(* Schneider Machine Expert - Basic project Maquina, file version 2.9.0.0 *)
(* ProjectInformations: Name=Nuevo proyecto *)

HARDWARE
  Cpu 0: TM221CE16T
  EthernetConfiguration: NetworkName=M221, IpAllocationMode=FixedAddress, IpAddress=192.168.0.10, SubnetMask=255.255.255.0
  SerialLineConfiguration: Baud=Baud19200, Parity=ParityEven, DataBits=DataBits8, StopBits=StopBits1, PhysicalMedium=PhysicalMediumRs485, TransmissionMode=TransmissionModeModbusRtu, SlaveId=1, Addressing=SlaveAddressing
  MastTask: UsePeriodScanMode=false, PeriodScan=100
  FastTask: Period=255
  CpuBehavior: StartingMode=StartAsPreviousState, AutoSaveRamOnEeprom=true, WatchdogPeriod=250

SYMBOLS  (address, symbol, comment, settings)
  %M1       INICIO_MANUAL  "start Manual"
  %M2       INICIO_AUTOM  "Automatico"
  %M3       STOP
  %M4       AUT_ARRIBA
  %M5       RESET  "Nueva medicion"
  %M6       RESET_MANUAL  "reset manual"
  %M8       TIEM_MUESTREO_ON
  %M9       SUBIR
  %M10      BAJAR  "Bajar_manual"
  %M12      BAJAR_AUTO  "Hab.Pulsos"
  %M13      GRAFICA  "Hab.Grafica"
  %M14      AUTOMA_ON
  %M15      HA_AUTOMATICO
  %M16      MANUAL_ON
  %M17      HA_MANUAL
  %M18      AUT_ABAJO
  %M19      SUBIR_AUTO
  %M20      ESTADO1
  %M21      ESTADO2
  %M22      ESTADO3
  %M23      ESTADO4
  %MW2      VALOR_MENOR
  %MW3      VALOR_MAYOR
  %MW4      MAYOR
  %MW8      TIEMPO_MUESTREO
  %MW11     DATOSGRAFICA
  %KW0      ESCA  [Value=10]
  %TM1        [Preset=10, Base=OneMilliSeconds]
  %TM2        [Preset=10, Base=OneMilliSeconds]
  %TM3        [Preset=10, Base=OneMilliSeconds]
  %I0.1     SEN_INFERIOR
  %I0.3     SEN_SUPERIOR
  %Q0.2     SENGIRO
  %IW0.1    CELDA  [Type=Type_0_10V, Scope=Scope_Normal, Minimum=0, Maximum=1000]
  %FREQGEN0 MOTOR  [PtoObject(RefInput=NotUsed, ZPhaseInput=NotUsed, ProbeInput=NotUsed), GlobalIndex=0, Type=FREQGEN, Preset=1, SignalFrequency=2000]
  %FREQGEN1 DATOS  [PtoObject(RefInput=NotUsed, ZPhaseInput=NotUsed, ProbeInput=NotUsed), GlobalIndex=1, Type=FREQGEN, TimeBase=OneMilliSeconds, Preset=1, SignalFrequency=200]

POU Nuevo POU
  (* SectionNumber=1 *)

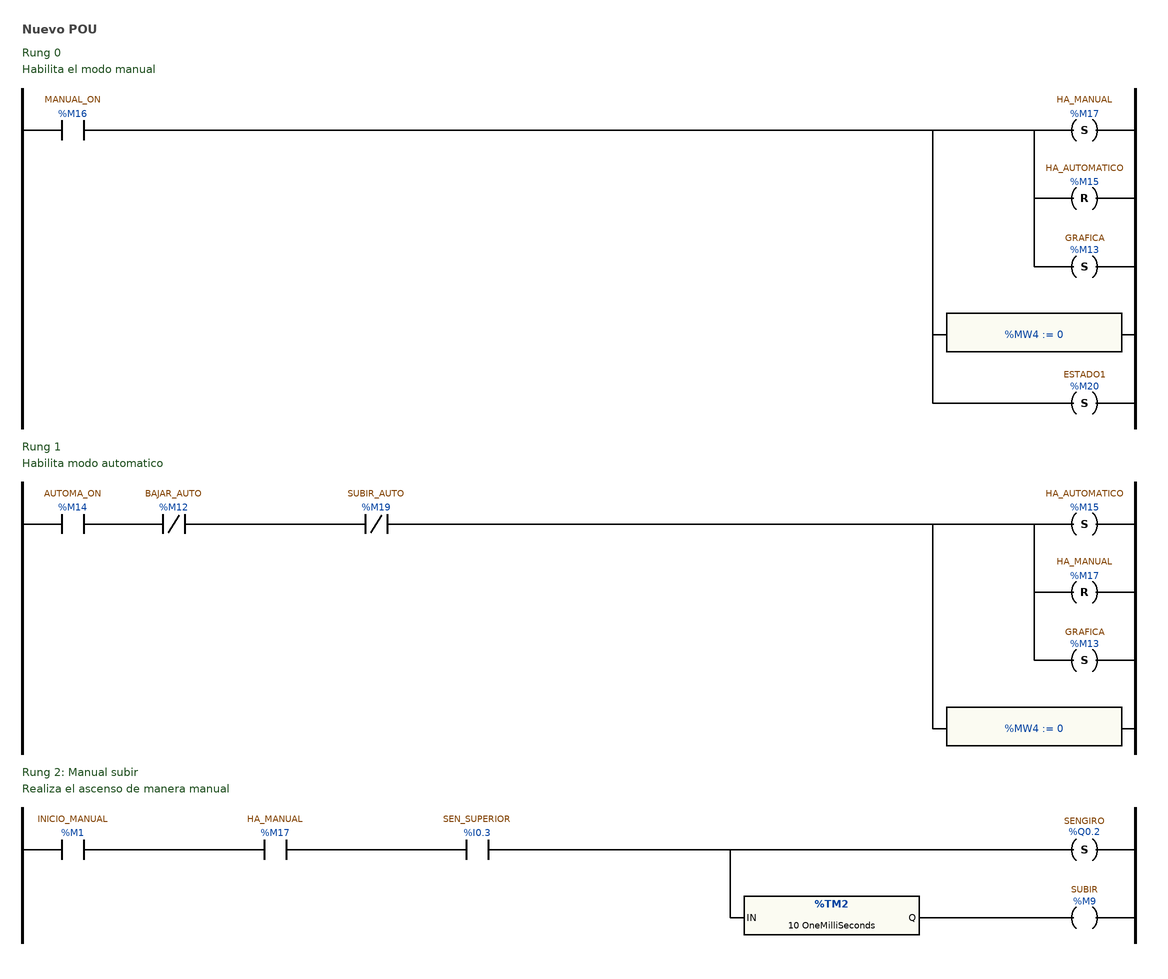

// Rung 0
// Habilita el modo manual
  LD %M16                 (* MANUAL_ON *)
  S %M17                  (* HA_MANUAL *)
  R %M15                  (* HA_AUTOMATICO *)
  S %M13                  (* GRAFICA *)
  [ %MW4 := 0 ]           (* MAYOR *)
  S %M20                  (* ESTADO1 *)
  // as ST:
  //   IF MANUAL_ON THEN HA_MANUAL := TRUE; END_IF;
  //   IF MANUAL_ON THEN HA_AUTOMATICO := FALSE; END_IF;
  //   IF MANUAL_ON THEN GRAFICA := TRUE; END_IF;
  //   IF MANUAL_ON THEN MAYOR := 0; END_IF;
  //   IF MANUAL_ON THEN ESTADO1 := TRUE; END_IF;

// Rung 1
// Habilita modo automatico
  LD %M14                 (* AUTOMA_ON *)
  ANDN %M12               (* BAJAR_AUTO *)
  ANDN %M19               (* SUBIR_AUTO *)
  S %M15                  (* HA_AUTOMATICO *)
  R %M17                  (* HA_MANUAL *)
  S %M13                  (* GRAFICA *)
  [ %MW4 := 0 ]           (* MAYOR *)
  // as ST:
  //   IF AUTOMA_ON AND NOT BAJAR_AUTO AND NOT SUBIR_AUTO THEN HA_AUTOMATICO := TRUE; END_IF;
  //   IF AUTOMA_ON AND NOT BAJAR_AUTO AND NOT SUBIR_AUTO THEN HA_MANUAL := FALSE; END_IF;
  //   IF AUTOMA_ON AND NOT BAJAR_AUTO AND NOT SUBIR_AUTO THEN GRAFICA := TRUE; END_IF;
  //   IF AUTOMA_ON AND NOT BAJAR_AUTO AND NOT SUBIR_AUTO THEN MAYOR := 0; END_IF;

// Rung 2: Manual subir
// Realiza el ascenso de manera manual
  LD 1
  MULTIFB
  LD 1
  AND %M1                 (* INICIO_MANUAL *)
  AND %M17                (* HA_MANUAL *)
  AND %I0.3               (* SEN_SUPERIOR *)
  ST %MW2009:X0
  LD %MW2009:X0
  S %Q0.2                 (* SENGIRO *)
  BLK %TM2
  LD %MW2009:X0
  IN
  OUT_BLK
  LD Q
  ST %M9                  (* SUBIR *)
  END_BLK
  MULTIFB
  // as ST:
  //   IF INICIO_MANUAL AND HA_MANUAL AND SEN_SUPERIOR THEN SENGIRO := TRUE; END_IF;
  //   %TM2(IN := INICIO_MANUAL AND HA_MANUAL AND SEN_SUPERIOR);
  //   SUBIR := %TM2.Q;

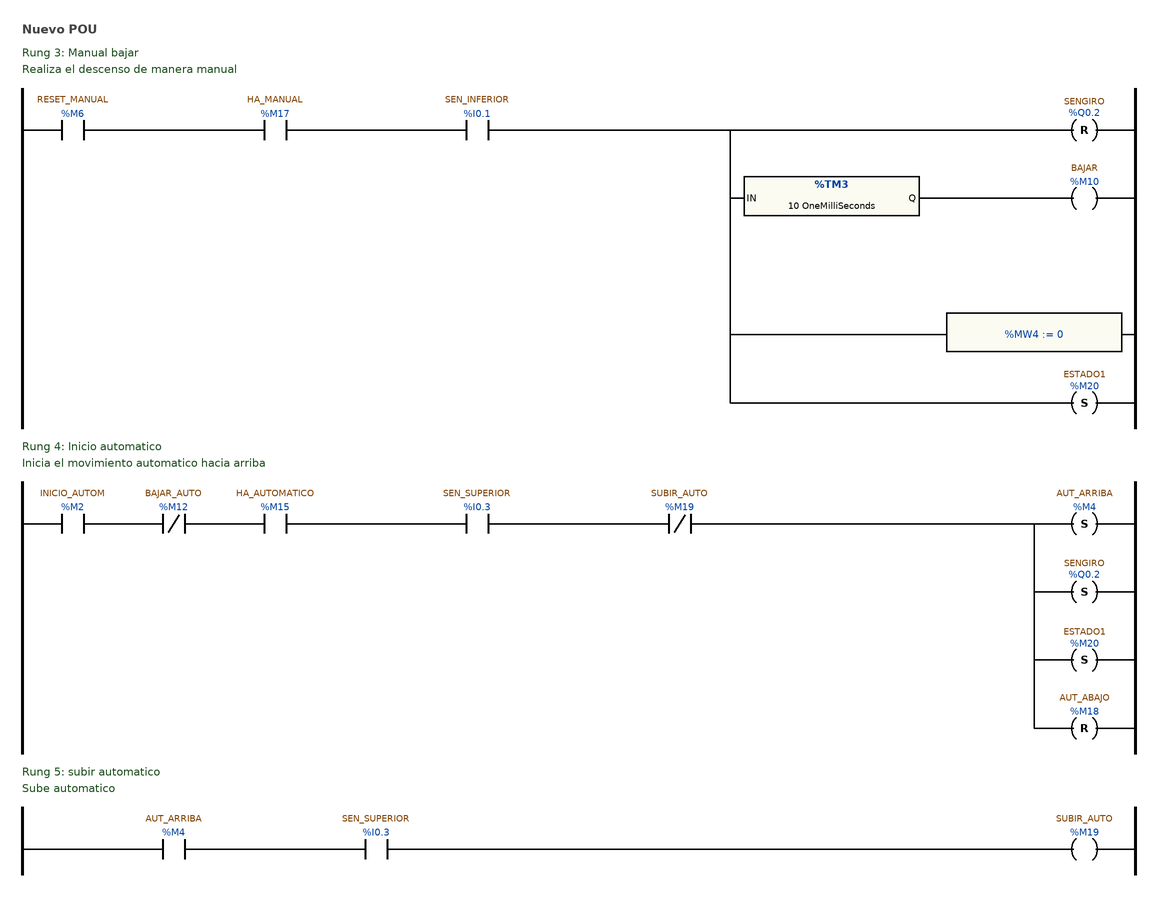

// Rung 3: Manual bajar
// Realiza el descenso de manera manual
  LD 1
  MULTIFB
  LD 1
  AND %M6                 (* RESET_MANUAL *)
  AND %M17                (* HA_MANUAL *)
  AND %I0.1               (* SEN_INFERIOR *)
  ST %MW2009:X0
  LD %MW2009:X0
  R %Q0.2                 (* SENGIRO *)
  BLK %TM3
  LD %MW2009:X0
  IN
  OUT_BLK
  LD Q
  ST %M10                 (* BAJAR *)
  END_BLK
  LD %MW2009:X0
  [ %MW4 := 0 ]           (* MAYOR *)
  S %M20                  (* ESTADO1 *)
  MULTIFB
  // as ST:
  //   IF RESET_MANUAL AND HA_MANUAL AND SEN_INFERIOR THEN SENGIRO := FALSE; END_IF;
  //   %TM3(IN := RESET_MANUAL AND HA_MANUAL AND SEN_INFERIOR);
  //   BAJAR := %TM3.Q;
  //   IF RESET_MANUAL AND HA_MANUAL AND SEN_INFERIOR THEN MAYOR := 0; END_IF;
  //   IF RESET_MANUAL AND HA_MANUAL AND SEN_INFERIOR THEN ESTADO1 := TRUE; END_IF;

// Rung 4: Inicio automatico
// Inicia el movimiento automatico hacia arriba
  LD %M2                  (* INICIO_AUTOM *)
  ANDN %M12               (* BAJAR_AUTO *)
  AND %M15                (* HA_AUTOMATICO *)
  AND %I0.3               (* SEN_SUPERIOR *)
  ANDN %M19               (* SUBIR_AUTO *)
  S %M4                   (* AUT_ARRIBA *)
  S %Q0.2                 (* SENGIRO *)
  S %M20                  (* ESTADO1 *)
  R %M18                  (* AUT_ABAJO *)
  // as ST:
  //   IF INICIO_AUTOM AND NOT BAJAR_AUTO AND HA_AUTOMATICO AND SEN_SUPERIOR AND NOT SUBIR_AUTO THEN AUT_ARRIBA := TRUE; END_IF;
  //   IF INICIO_AUTOM AND NOT BAJAR_AUTO AND HA_AUTOMATICO AND SEN_SUPERIOR AND NOT SUBIR_AUTO THEN SENGIRO := TRUE; END_IF;
  //   IF INICIO_AUTOM AND NOT BAJAR_AUTO AND HA_AUTOMATICO AND SEN_SUPERIOR AND NOT SUBIR_AUTO THEN ESTADO1 := TRUE; END_IF;
  //   IF INICIO_AUTOM AND NOT BAJAR_AUTO AND HA_AUTOMATICO AND SEN_SUPERIOR AND NOT SUBIR_AUTO THEN AUT_ABAJO := FALSE; END_IF;

// Rung 5: subir automatico
// Sube automatico
  LD %M4                  (* AUT_ARRIBA *)
  AND %I0.3               (* SEN_SUPERIOR *)
  ST %M19                 (* SUBIR_AUTO *)
  // as ST:
  //   SUBIR_AUTO := AUT_ARRIBA AND SEN_SUPERIOR;

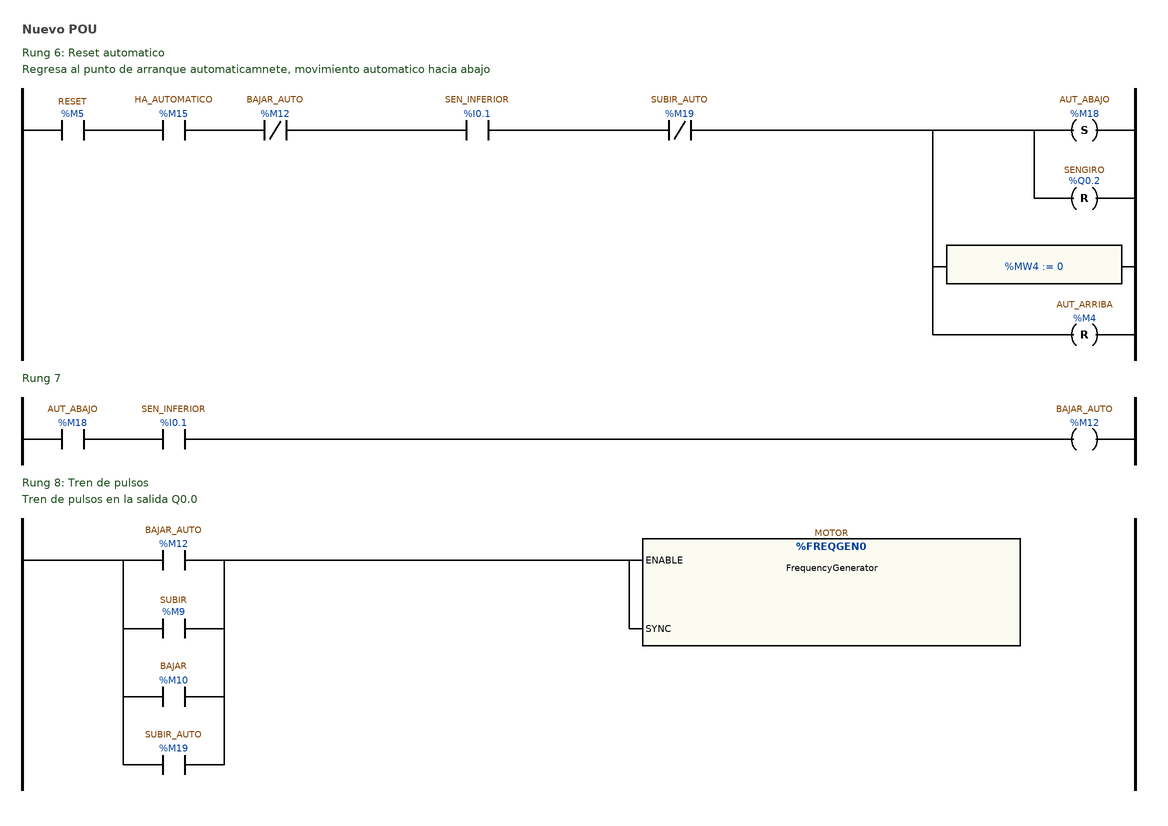

// Rung 6: Reset automatico
// Regresa al punto de arranque automaticamnete, movimiento automatico hacia abajo
  LD %M5                  (* RESET *)
  AND %M15                (* HA_AUTOMATICO *)
  ANDN %M12               (* BAJAR_AUTO *)
  AND %I0.1               (* SEN_INFERIOR *)
  ANDN %M19               (* SUBIR_AUTO *)
  S %M18                  (* AUT_ABAJO *)
  R %Q0.2                 (* SENGIRO *)
  [ %MW4 := 0 ]           (* MAYOR *)
  R %M4                   (* AUT_ARRIBA *)
  // as ST:
  //   IF RESET AND HA_AUTOMATICO AND NOT BAJAR_AUTO AND SEN_INFERIOR AND NOT SUBIR_AUTO THEN AUT_ABAJO := TRUE; END_IF;
  //   IF RESET AND HA_AUTOMATICO AND NOT BAJAR_AUTO AND SEN_INFERIOR AND NOT SUBIR_AUTO THEN SENGIRO := FALSE; END_IF;
  //   IF RESET AND HA_AUTOMATICO AND NOT BAJAR_AUTO AND SEN_INFERIOR AND NOT SUBIR_AUTO THEN MAYOR := 0; END_IF;
  //   IF RESET AND HA_AUTOMATICO AND NOT BAJAR_AUTO AND SEN_INFERIOR AND NOT SUBIR_AUTO THEN AUT_ARRIBA := FALSE; END_IF;

// Rung 7
  LD %M18                 (* AUT_ABAJO *)
  AND %I0.1               (* SEN_INFERIOR *)
  ST %M12                 (* BAJAR_AUTO *)
  // as ST:
  //   BAJAR_AUTO := AUT_ABAJO AND SEN_INFERIOR;

// Rung 8: Tren de pulsos
// Tren de pulsos en la salida Q0.0
  BLK %FREQGEN0           (* MOTOR *)
  LD 1
  AND( %M12               (* BAJAR_AUTO *)
  OR %M9                  (* SUBIR *)
  OR %M10                 (* BAJAR *)
  OR %M19                 (* SUBIR_AUTO *)
  )
  ENABLE
  SYNC
  END_BLK
  // as ST:
  //   MOTOR(ENABLE := BAJAR_AUTO OR SUBIR OR BAJAR OR SUBIR_AUTO, SYNC := BAJAR_AUTO OR SUBIR OR BAJAR OR SUBIR_AUTO);

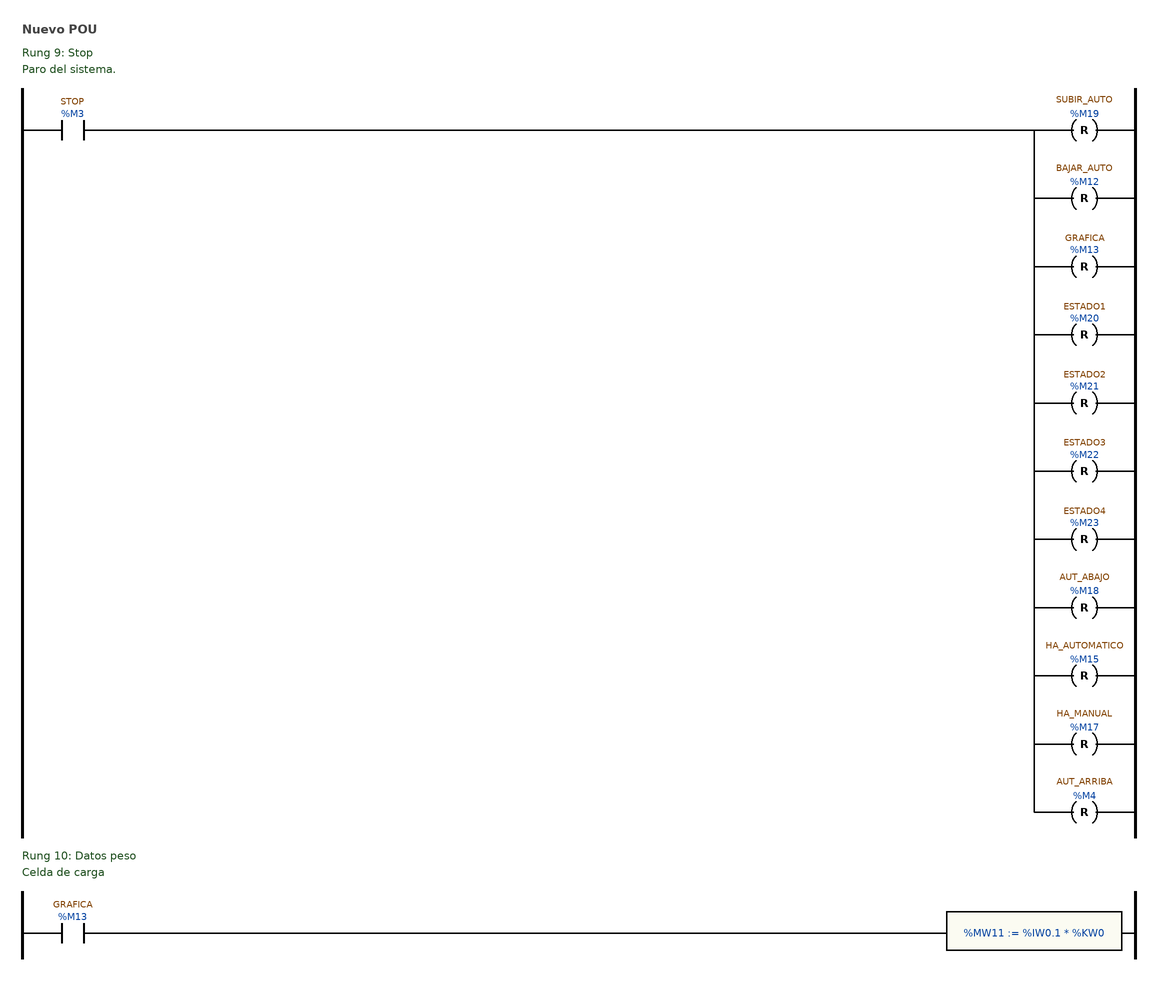

// Rung 9: Stop
// Paro del sistema.
  LD %M3                  (* STOP *)
  R %M19                  (* SUBIR_AUTO *)
  R %M12                  (* BAJAR_AUTO *)
  R %M13                  (* GRAFICA *)
  R %M20                  (* ESTADO1 *)
  R %M21                  (* ESTADO2 *)
  R %M22                  (* ESTADO3 *)
  R %M23                  (* ESTADO4 *)
  R %M18                  (* AUT_ABAJO *)
  R %M15                  (* HA_AUTOMATICO *)
  R %M17                  (* HA_MANUAL *)
  R %M4                   (* AUT_ARRIBA *)
  // as ST:
  //   IF STOP THEN SUBIR_AUTO := FALSE; END_IF;
  //   IF STOP THEN BAJAR_AUTO := FALSE; END_IF;
  //   IF STOP THEN GRAFICA := FALSE; END_IF;
  //   IF STOP THEN ESTADO1 := FALSE; END_IF;
  //   IF STOP THEN ESTADO2 := FALSE; END_IF;
  //   IF STOP THEN ESTADO3 := FALSE; END_IF;
  //   IF STOP THEN ESTADO4 := FALSE; END_IF;
  //   IF STOP THEN AUT_ABAJO := FALSE; END_IF;
  //   IF STOP THEN HA_AUTOMATICO := FALSE; END_IF;
  //   IF STOP THEN HA_MANUAL := FALSE; END_IF;
  //   IF STOP THEN AUT_ARRIBA := FALSE; END_IF;

// Rung 10: Datos peso
// Celda de carga
  LD %M13                 (* GRAFICA *)
  [ %MW11 := %IW0.1 * %KW0 ](* DATOSGRAFICA, CELDA, ESCA *)
  // as ST:
  //   IF GRAFICA THEN DATOSGRAFICA := CELDA * ESCA; END_IF;

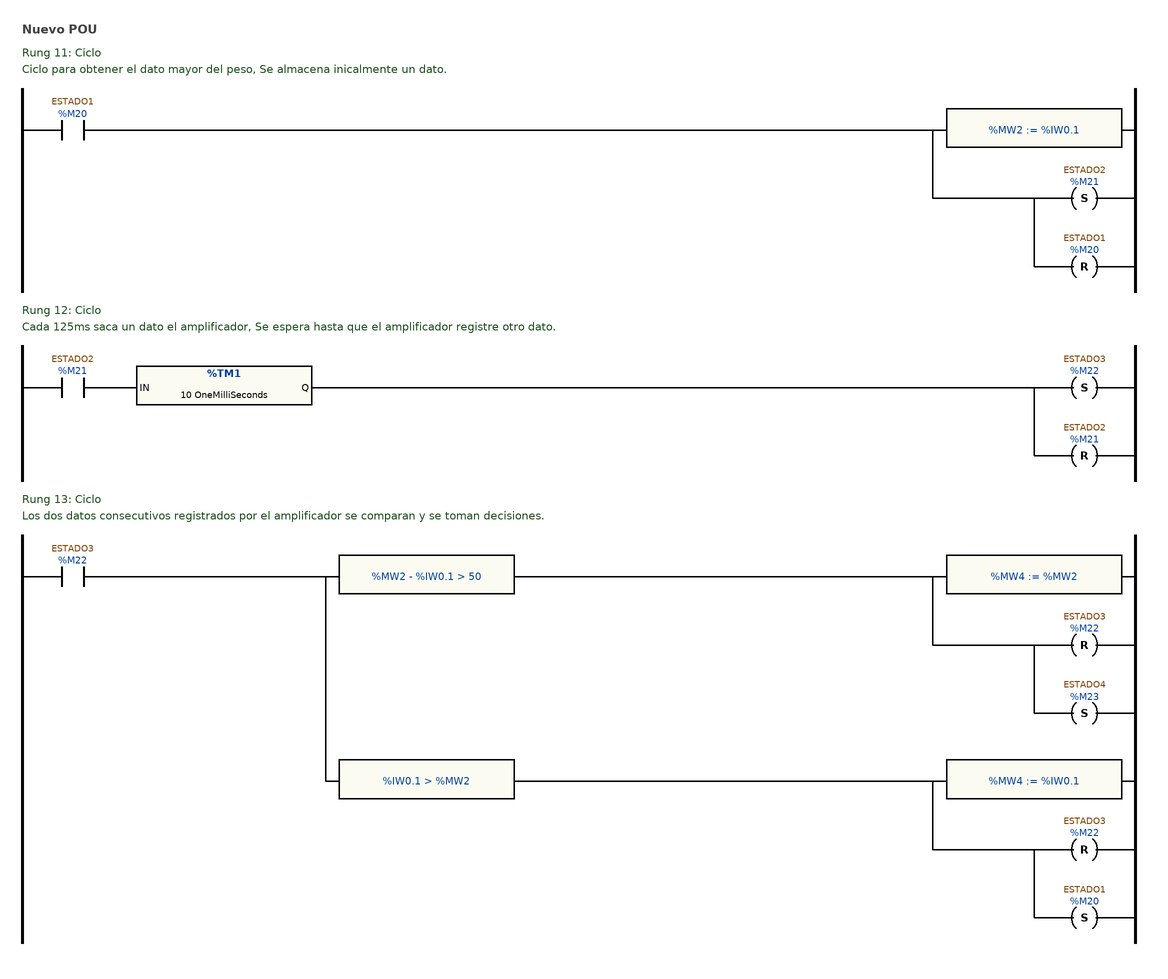

// Rung 11: Ciclo
// Ciclo para obtener el dato mayor del peso, Se almacena inicalmente un dato.
  LD %M20                 (* ESTADO1 *)
  [ %MW2 := %IW0.1 ]      (* VALOR_MENOR, CELDA *)
  S %M21                  (* ESTADO2 *)
  R %M20                  (* ESTADO1 *)
  // as ST:
  //   IF ESTADO1 THEN VALOR_MENOR := CELDA; END_IF;
  //   IF ESTADO1 THEN ESTADO2 := TRUE; END_IF;
  //   IF ESTADO1 THEN ESTADO1 := FALSE; END_IF;

// Rung 12: Ciclo
// Cada 125ms saca un dato el amplificador, Se espera hasta que el amplificador registre otro dato.
  BLK %TM1
  LD %M21                 (* ESTADO2 *)
  IN
  OUT_BLK
  LD Q
  S %M22                  (* ESTADO3 *)
  R %M21                  (* ESTADO2 *)
  END_BLK
  // as ST:
  //   %TM1(IN := ESTADO2);
  //   IF %TM1.Q THEN ESTADO3 := TRUE; END_IF;
  //   IF %TM1.Q THEN ESTADO2 := FALSE; END_IF;

// Rung 13: Ciclo
// Los dos datos consecutivos registrados por el amplificador se comparan y se toman decisiones.
  LD %M22                 (* ESTADO3 *)
  MPS
  AND [ %MW2 - %IW0.1 > 50 ](* VALOR_MENOR, CELDA *)
  [ %MW4 := %MW2 ]        (* MAYOR, VALOR_MENOR *)
  R %M22                  (* ESTADO3 *)
  S %M23                  (* ESTADO4 *)
  MPP
  AND [ %IW0.1 > %MW2 ]   (* CELDA, VALOR_MENOR *)
  [ %MW4 := %IW0.1 ]      (* MAYOR, CELDA *)
  R %M22                  (* ESTADO3 *)
  S %M20                  (* ESTADO1 *)
  // as ST:
  //   IF ESTADO3 AND VALOR_MENOR - CELDA > 50 THEN MAYOR := VALOR_MENOR; END_IF;
  //   _t1 := ESTADO3;
  //   _t2 := ESTADO3 AND VALOR_MENOR - CELDA > 50;
  //   IF _t2 THEN ESTADO3 := FALSE; END_IF;
  //   IF _t2 THEN ESTADO4 := TRUE; END_IF;
  //   IF _t1 AND CELDA > VALOR_MENOR THEN MAYOR := CELDA; END_IF;
  //   IF _t1 AND CELDA > VALOR_MENOR THEN ESTADO3 := FALSE; END_IF;
  //   IF _t1 AND CELDA > VALOR_MENOR THEN ESTADO1 := TRUE; END_IF;

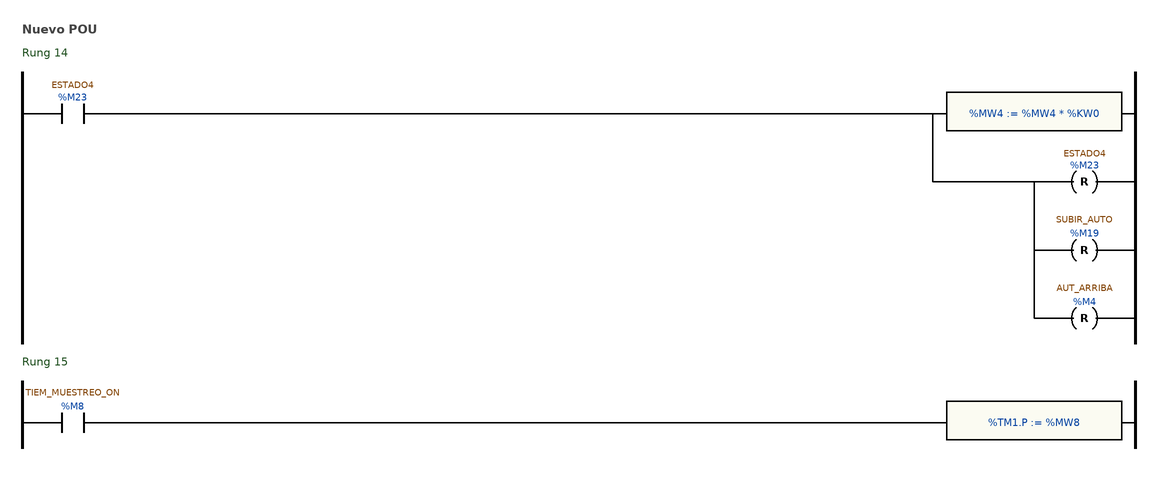

// Rung 14
  LD %M23                 (* ESTADO4 *)
  [ %MW4 := %MW4 * %KW0 ] (* MAYOR, MAYOR, ESCA *)
  R %M23                  (* ESTADO4 *)
  R %M19                  (* SUBIR_AUTO *)
  R %M4                   (* AUT_ARRIBA *)
  // as ST:
  //   IF ESTADO4 THEN MAYOR := MAYOR * ESCA; END_IF;
  //   _t1 := ESTADO4;
  //   IF _t1 THEN ESTADO4 := FALSE; END_IF;
  //   IF _t1 THEN SUBIR_AUTO := FALSE; END_IF;
  //   IF _t1 THEN AUT_ARRIBA := FALSE; END_IF;

// Rung 15
  LD %M8                  (* TIEM_MUESTREO_ON *)
  [ %TM1.P := %MW8 ]      (* TIEMPO_MUESTREO *)
  // as ST:
  //   IF TIEM_MUESTREO_ON THEN %TM1.P := TIEMPO_MUESTREO; END_IF;
